// TIA Portal V19 export
TYPE "LUC_typeSignalStackByStatus"
// Stack Light Signals by Bool
// stored: Access Published
   STRUCT
      redSolid { ExternalWritable := 'False'} : Bool;   // Red light solid
      redFlashing { ExternalWritable := 'False'} : Bool;   // Red light flashing
      yellowSolid { ExternalWritable := 'False'} : Bool;   // Yellow light solid
      yellowFlashing { ExternalWritable := 'False'} : Bool;   // Yellow light flashing
      blueSolid { ExternalWritable := 'False'} : Bool;   // Blue light solid
      blueFlashing { ExternalWritable := 'False'} : Bool;   // Blue light flashing
      greenSolid { ExternalWritable := 'False'} : Bool;   // Green light solid
      greenFlashing { ExternalWritable := 'False'} : Bool;   // Green light flashing
      hornSolid { ExternalWritable := 'False'} : Bool;   // Horn solid
      hornFlashing { ExternalWritable := 'False'} : Bool;   // Horn flashing
      whiteSolid { ExternalWritable := 'False'} : Bool;   // White light solid
      whiteFlashing { ExternalWritable := 'False'} : Bool;   // White light flashing
      user1Solid { ExternalWritable := 'False'} : Bool;   // User defined light solid
      user1Flashing { ExternalWritable := 'False'} : Bool;   // User defined light flashing
      user2Solid { ExternalWritable := 'False'} : Bool;   // User defined light solid
      user2Flashing { ExternalWritable := 'False'} : Bool;   // User defined light flashing
   END_STRUCT;
END_TYPE
